{attribute addProperty BoxType "EP4378-1022-0017"}
{attribute addProperty Id "InputAT %I*BOOL81"}
{attribute addProperty CRC "3836671390"}
{attribute addProperty SizeInBites "8"}
{attribute addProperty SizeInBytes "1"}
TYPE DI_X05_Pin4_Input_E4AEF59E :
STRUCT
	{attribute addProperty Name "Input"}
	Input AT %I* : BOOL;
END_STRUCT
END_TYPE

(* stored: Version 1.2.0.0, ProductVersion 3.1.4024.9
   DUT DI_X05_Pin4_Input_E4AEF59E: Id {8d5f8967-59cd-41c2-a72d-fd42f90703d0} *)
